{attribute 'qualified_only'}
VAR_GLOBAL
	MessageNo	: UDINT := 1;
	
END_VAR

(* stored: Version 1.1.0.1, ProductVersion 3.1.4024.12
   GVL TcpIpCommVars: Id {bed03919-34a6-4327-ace1-019cf37847e3} *)
